PROGRAM MQTTCommunication
VAR_INPUT
	fbMqttClient    : FB_IotMqttClient;
END_VAR
VAR
    bSetParameter   : BOOL := TRUE;
    bConnect        : BOOL := TRUE;
	(* published message *)
    sTopicPub   : STRING(255) := 'STELLA';
    sPayloadPub : STRING(255);
	epos : INT;
//	bPublished:		BOOL;
	(* received message *)
    bSubscribed    : BOOL;
    sTopicSub      : STRING(255) := 'STELLA/Telemetry/SET';
    {attribute 'TcEncoding':='UTF-8'}
    sTopicRcv      : STRING(255);
    {attribute 'TcEncoding':='UTF-8'}
    sPayloadRcv    : STRING(255);
	parameter:		STRING(255);
	value:			LREAL;
    fbMessageQueue : FB_IotMqttMessageQueue;
    fbMessage      : FB_IotMqttMessage;
END_VAR

(*
MQTT Communication section

Source:
https://infosys.beckhoff.com/english.php?content=../content/1033/tf6701_tc3_iot_communication_mqtt/3518541195.html&id=

*)

// set the parameters once
IF bSetParameter THEN
    bSetParameter               := FALSE;
    fbMqttClient.sHostName      := 'sky.stella.iac.es';
    fbMqttClient.nHostPort      := 1883;
    fbMqttClient.sClientId      := 'STELLAroofPLCnew'; 
    fbMqttClient.sTopicPrefix   := ''; 
	fbMqttClient.nKeepAlive     := 60; 
//  fbMqttClient.sUserName      := ;
//  fbMqttClient.sUserPassword  := ; 
//  fbMqttClient.stWill         := ; 
//  fbMqttClient.stTLS          := ;
    fbMqttClient.ipMessageQueue := fbMessageQueue;
END_IF

// connect to the client
fbMqttClient.Execute(bConnect);

IF fbMqttClient.bConnected THEN
    IF NOT bSubscribed THEN
        bSubscribed := fbMqttClient.Subscribe(sTopic:=sTopicSub, eQoS:=TcIotMqttQos.AtMostOnceDelivery);
    END_IF
END_IF
(*
// receive queued messages
IF fbMessageQueue.nQueuedMessages > 0 THEN
    IF fbMessageQueue.Dequeue(fbMessage:=fbMessage) THEN
        fbMessage.GetTopic(pTopic:=ADR(sTopicRcv), nTopicSize:=SIZEOF(sTopicRcv) );
        fbMessage.GetPayload(pPayload:=ADR(sPayloadRcv), nPayloadSize:=SIZEOF(sPayloadRcv), bSetNullTermination:=FALSE);
		IF sTopicRcv = 'RoboTel/Telescope/SET' THEN
			epos := FIND(sPayloadRcv, '=');
			parameter := LEFT(sPayloadRcv, epos-1);
			value := STRING_TO_LREAL(DELETE(sPayloadRcv, epos+2, 1));
			IF parameter = 'Declination' THEN
				TelescopeControl.de := value;
			ELSIF parameter = 'RightAscension' THEN
				TelescopeControl.ra := value;
			END_IF
		END_IF
    END_IF
END_IF
*)

END_PROGRAM

(* stored: Version 1.1.0.1, ProductVersion 3.1.4024.9
   POU MQTTCommunication: Id {7764f620-4215-4717-9686-e3cbacd7309d}, SpecialFunc None *)
